% RSLogix 500 project HOURMETER.RSS, saved by version 8.30.00.16 %
PROJECT "UNTITLED"    % processor: Bul.1763 MicroLogix 1100 Series B %

PROGRAM FILES
  LAD 2 "MAIN"  3 rungs
  LAD 3 "INPUT"  3 rungs
  LAD 4 "HOURMETER"  7 rungs

DATA FILES
  O0 OUTPUT  4 elements
  I1 INPUT  6 elements
  S2 STATUS  66 elements
  B3 BINARY  2 elements
  T4 TIMER  1 elements
  C5 COUNTER  1 elements
  R6 CONTROL  1 elements
  N7 INTEGER  10 elements
  F8 FLOAT  1 elements

LADDER 2 "MAIN"
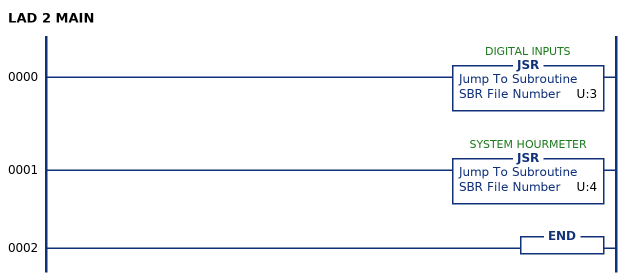
% Rung: 0 %
SOR JSR U:3 EOR
%   U:3  "DIGITAL INPUTS" %
% Rung: 1 %
SOR JSR U:4 EOR
%   U:4  "SYSTEM HOURMETER" %
% Rung: 2 %
SOR END EOR

LADDER 3 "INPUT"
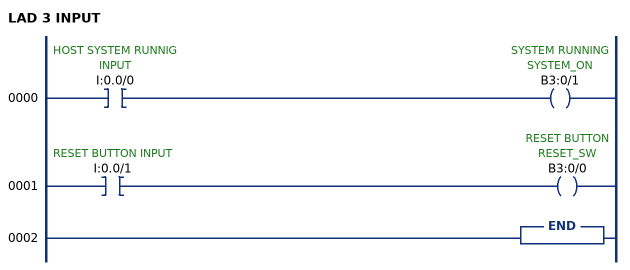
% Rung: 0 %
SOR XIC I:0.0/0 OTE B3:0/1 EOR
%   I:0.0/0  "HOST SYSTEM RUNNIG INPUT" %
%   B3:0/1  SYSTEM_ON  "SYSTEM RUNNING" %
% Rung: 1 %
SOR XIC I:0.0/1 OTE B3:0/0 EOR
%   I:0.0/1  "RESET BUTTON INPUT" %
%   B3:0/0  RESET_SW  "RESET BUTTON" %
% Rung: 2 %
SOR END EOR

LADDER 4 "HOURMETER"
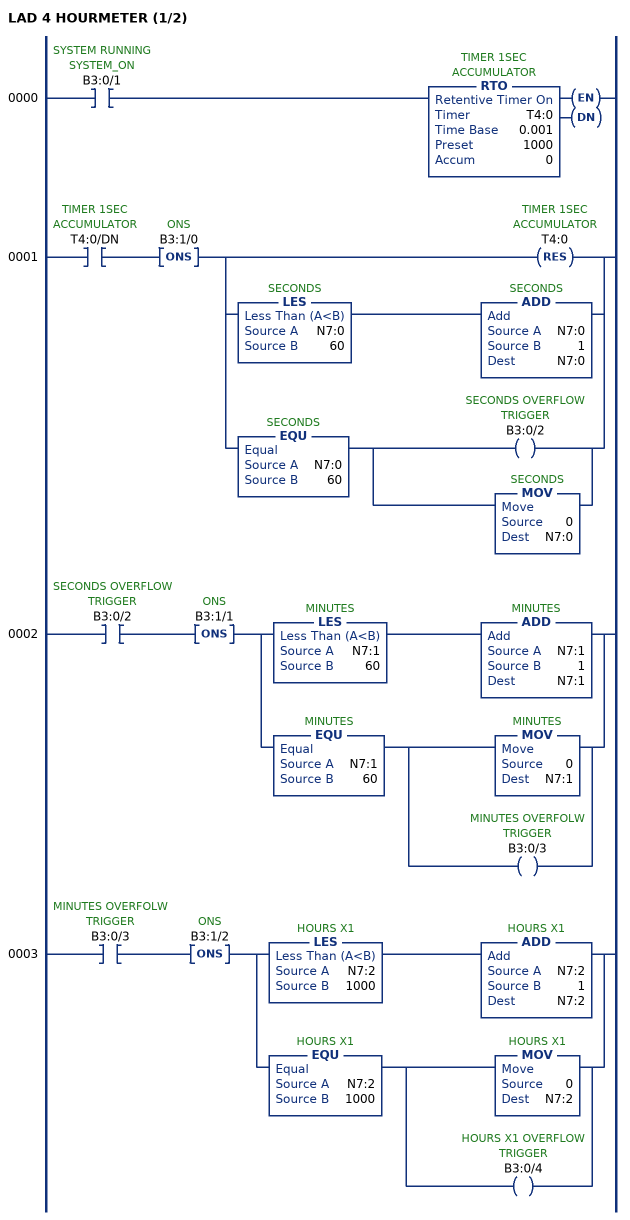
% Rung: 0 %
SOR XIC B3:0/1 RTO T4:0 0.001 1000 0 EOR
%   B3:0/1  SYSTEM_ON  "SYSTEM RUNNING" %
%   T4:0  "TIMER 1SEC ACCUMULATOR" %
% Rung: 1 %
SOR XIC T4:0/DN ONS B3:1/0 BST RES T4:0 NXB LES N7:0 60 ADD N7:0 1 N7:0 NXB EQU N7:0 60 BST OTE B3:0/2 NXB MOV 0 N7:0 BND BND EOR
%   T4:0  "TIMER 1SEC ACCUMULATOR" %
%   B3:1/0  "ONS" %
%   N7:0  "SECONDS" %
%   B3:0/2  "SECONDS OVERFLOW TRIGGER" %
% Rung: 2 %
SOR XIC B3:0/2 ONS B3:1/1 BST LES N7:1 60 ADD N7:1 1 N7:1 NXB EQU N7:1 60 BST MOV 0 N7:1 NXB OTE B3:0/3 BND BND EOR
%   B3:0/2  "SECONDS OVERFLOW TRIGGER" %
%   B3:1/1  "ONS" %
%   N7:1  "MINUTES" %
%   B3:0/3  "MINUTES OVERFOLW TRIGGER" %
% Rung: 3 %
SOR XIC B3:0/3 ONS B3:1/2 BST LES N7:2 1000 ADD N7:2 1 N7:2 NXB EQU N7:2 1000 BST MOV 0 N7:2 NXB OTE B3:0/4 BND BND EOR
%   B3:0/3  "MINUTES OVERFOLW TRIGGER" %
%   B3:1/2  "ONS" %
%   N7:2  "HOURS X1" %
%   B3:0/4  "HOURS X1 OVERFLOW TRIGGER" %

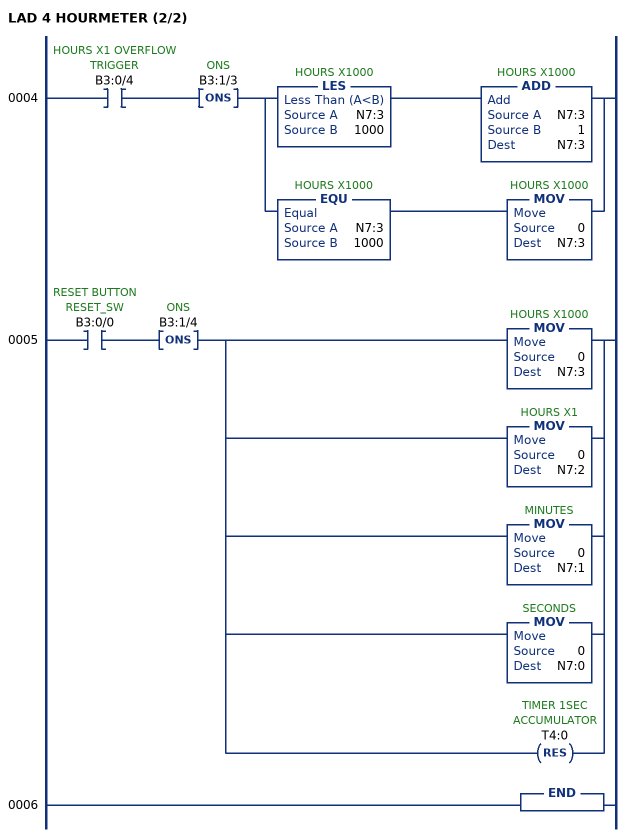
% Rung: 4 %
SOR XIC B3:0/4 ONS B3:1/3 BST LES N7:3 1000 ADD N7:3 1 N7:3 NXB EQU N7:3 1000 MOV 0 N7:3 BND EOR
%   B3:0/4  "HOURS X1 OVERFLOW TRIGGER" %
%   B3:1/3  "ONS" %
%   N7:3  "HOURS X1000" %
% Rung: 5 %
SOR XIC B3:0/0 ONS B3:1/4 BST MOV 0 N7:3 NXB MOV 0 N7:2 NXB MOV 0 N7:1 NXB MOV 0 N7:0 NXB RES T4:0 BND EOR
%   B3:0/0  RESET_SW  "RESET BUTTON" %
%   B3:1/4  "ONS" %
%   N7:3  "HOURS X1000" %
%   N7:2  "HOURS X1" %
%   N7:1  "MINUTES" %
%   N7:0  "SECONDS" %
%   T4:0  "TIMER 1SEC ACCUMULATOR" %
% Rung: 6 %
SOR END EOR

DATA TABLE (non-zero values as saved)
DATA T4
% .PRE .ACC %
% T4:0 % 1000 0
